{attribute 'qualified_only'}
VAR_GLOBAL
	//Zmienne obslugi bledow
	bError										: BOOL;														// Zmienna ogolna wystapienia bledu                                                                         							
	udiErrorID									: UDINT;													// Kod bledu 	
	sErrorDescription1							: STRING(200);												// Opis bledu 1
	sErrorDescription2							: STRING(200);												// Opis bledu 2
	sStationInError								: STRING(200);												// Nazwa stacji w bledzie
                                                 
                                                                        	

	tonResettingTime							: TON;														// Licznik odliczacy czas wykonywania procedury resetu
	
	iStep										: INT;														// Krok proedury czytania bledow 	

END_VAR


VAR_GLOBAL CONSTANT
	iErrorStructuresNumber						: INT					:= 9;								// Liczba strukur bledow stacji  w tym strukura bledow globalnych
END_VAR

(* stored: Version 1.1.0.1, FileIdentifier ba7a476d28b344ea294beff788237f7380033e62, FileSignature 293bdf63fb058e4de1c76cc11227d2e25d77d6d86a5cd7933f1f317085ac39d5ffee6bb720a324467d1668f90dfab5a226e882ddb796b637842b51220e28b003a12ec77bd069415a5bb6306aa4db059252a138eb014fdffd73fb1bb8f0240134f49223238d9a83f127485eb13a3797368237310b3770cdbaa6e99ef68d809e20c262af016dd6b68aacd6e829456ecd637e5fac9320004234349d64b2295d985aedd40e09c7d3a04c5d05504ed866de2f8ded4aee5f2dd610b719259e50045359257a6348ba7dc7361caacc31611f581ede62b2e5a8fb20656f057c5e5d940cbe7d447dc1e57a4b2c198171dfb8feb53acf87c9b69b5db4c8606c3f0150b93bf0
   GVL GVL_ErrorHandling: Id {fdb0a21e-0864-48c1-9390-6d8e4aa88279} *)
